{attribute 'qualified_only' := ''}
{attribute 'strict' := ''}
TYPE E_Pose :
(
	One := 0,
	Two := 1,
	Three := 2,
	Four := 3,
	Five := 4
);
END_TYPE

(* stored: Version 1.1.0.1
   DUT E_Pose: Id {b79aef52-6212-478e-b00a-eac3efda95a0} *)
